// TwinCAT 3 PLC project PlcAxis
// ProgramVersion: 3.1.4024.0
// project tree:
//   POUs/ I_Drivable.TcIO, FB_Axis.TcPOU, MAIN.TcPOU

// ---- POUs/I_Drivable.TcIO
INTERFACE I_Drivable

END_INTERFACE

// ---- POUs/FB_Axis.TcPOU
FUNCTION_BLOCK FB_Axis IMPLEMENTS I_Drivable
VAR
    bRunning : BOOL;
END_VAR

METHOD Start
bRunning := TRUE;
END_METHOD

END_FUNCTION_BLOCK

// ---- POUs/MAIN.TcPOU
PROGRAM MAIN
VAR
    axis : FB_Axis;
END_VAR

axis.Start();

END_PROGRAM
